{attribute 'pack_mode' := '2'}
TYPE ST_XPU_STATE :
STRUCT
  Init            : E_XPU_INIT;
  State           : E_XPU_STATE;
  Check           : E_XPU_CHECK;  // cyclic check result
  DcLink          : BIT;          // power all motor modules is ON
END_STRUCT
END_TYPE

(* stored: Version 1.1.0.1
   DUT ST_XPU_STATE: Id {2c71796c-fe96-4c32-955b-e39f01a1f8ac} *)
